// TwinCAT 3 PLC project factorialPLC
// ProgramVersion: 3.1.4024.0
// libraries:
//   Tc2_Standard, * (Beckhoff Automation GmbH)
//   Tc2_System, * (Beckhoff Automation GmbH)
//   Tc2_Utilities, * (Beckhoff Automation GmbH)
//   Tc3_Module, * (Beckhoff Automation GmbH)
// project tree:
//   / PlcTask.TcTTO
//   POUs/ F_factorial.TcPOU, MAIN.TcPOU

CONFIGURATION factorialPLC
    RESOURCE PLC ON TwinCAT3
        TASK PlcTask(INTERVAL := T#10ms, PRIORITY := 23);
        PROGRAM MAIN WITH PlcTask : MAIN;
    END_RESOURCE
END_CONFIGURATION

// ---- POUs/MAIN.TcPOU
PROGRAM MAIN
VAR
	fbProfiler : Profiler;
	stProfilerData : PROFILERSTRUCT;
	numFactorial : ULINT;
END_VAR

fbProfiler(START := TRUE, RESET := FALSE);
F_factorial(n := numFactorial);
fbProfiler(START := FALSE);
stProfilerData := fbProfiler.DATA;

END_PROGRAM

// ---- POUs/F_factorial.TcPOU
FUNCTION F_factorial : ULINT
VAR_INPUT
	n : ULINT;
END_VAR
VAR
	tempFact : ULINT;
	i : ULINT;
END_VAR

tempFact := 1;
FOR i := 1 TO n BY 1 DO
	tempFact := i * tempFact;
END_FOR
F_factorial := tempFact;

END_FUNCTION
